Staubli VAL3: Control_BottomS.pgx

public program Control_BottomS(string x_sBottomList)
  local string l_sBottomList[8]
  local bool l_bRes
begin

  call Str_SplitComma(l_bRes,x_sBottomList,l_sBottomList)
  if !l_bRes
    return
  endIf

call Control_Bottom(l_sBottomList)

end
